INTERFACE ITF_DigIn

PROPERTY ActualValue : BOOL
GET
END_GET
SET
END_SET
END_PROPERTY

PROPERTY FallingEdge : BOOL
GET
END_GET
SET
END_SET
END_PROPERTY

METHOD FB_init : BOOL
VAR_INPUT
	bInitRetains : BOOL; // if TRUE, the retain variables are initialized (warm start / cold start)
	bInCopyCode : BOOL;  // if TRUE, the instance afterwards gets moved into the copy code (online change)
END_VAR
END_METHOD

METHOD Force : BOOL
VAR_INPUT
	ForceValue : BOOL;
END_VAR
END_METHOD

METHOD ResetForce : BOOL
VAR_INPUT
END_VAR
END_METHOD

PROPERTY RisingEdge : BOOL
GET
END_GET
SET
END_SET
END_PROPERTY

END_INTERFACE

(* stored: Version 1.1.0.1, ProductVersion 3.1.4024.12
   Itf ITF_DigIn: Id {d6b083e4-706c-4235-919b-aa75848fe5ee}
   Folder Methods: Id {b886cc7d-444c-4018-a3d6-76ab11388afc}
   Folder Properties: Id {2fbfc247-2638-4066-88ce-b49a95e9a6c7}
   Property ActualValue: Id {60285ae5-b17f-4dc6-a4a7-22d69b4f5780}
   Get Get: Id {b1c40a2d-1c45-4abf-8702-275857beabf5}
   Set Set: Id {fc6df2c5-85c3-493a-a6f8-e3979125c889}
   Property FallingEdge: Id {e2ed51f1-31f3-47ce-981f-e52582876816}
   Get Get: Id {827d52ac-5d39-4228-97ef-73d3ec5c42a5}
   Set Set: Id {4f0e44d0-3d0a-4eae-b788-b4e28a1ab847}
   Method FB_init: Id {b3ad9bdb-5fe8-46fd-944c-8871e42f26df}
   Method Force: Id {9e1bf86f-bb97-4ead-8f3b-4dc2cc39ff3a}
   Method ResetForce: Id {013d1784-ff58-48f7-b9b5-3897f10bb995}
   Property RisingEdge: Id {4d9affa7-bc00-4efa-8d85-2596e49ea2ce}
   Get Get: Id {b4f459de-d3c4-4351-835a-1f7158d6f56f}
   Set Set: Id {d0a298fc-0930-467a-80fc-13a1cfd6c46d} *)
